// Block: RTrk

DATA_BLOCK RTrk
VERSION : 0.1
   NON_RETAIN
   VAR
      Last_RTrk_ID : DInt;
   END_VAR

BEGIN
   // No initialization required
END_DATA_BLOCK
